TYPE AxHomingParameters :
STRUCT
	TipoHoming : INT; //Tipologia di homing da eseguire
	InvertiDirezione : BOOL; //FALSE=Direzione NEgativa, TRUE=Direzione positiva
END_STRUCT
END_TYPE

(* stored: Version 1.1.0.1, ProductVersion 3.1.4024.11
   DUT AxHomingParameters: Id {84665482-50d5-4863-8ca8-70849762d39d} *)
